(* IEC 61131-3 sources: ATCMcontrol_Engineering/src/Target/ATHW119/Libs/ATCM_System2, 31 files *)

(* ---- EVT_GetEvent.st ---- *)
(*
 * ATCMControl Embedded - System Library
 * ----------------------------------------------------------------------------
 *

 *)

(*[[
    UserURL= "ATCMfile:EVT_GetEvent.htm"
]]*)

(* EVT_GetEvent
 * ----------------------------------------------------------------------------
 * Gets the last event whiched caused the execution of the corresponding event
 * driven task.
 *
 * in   sTask       Task name.
 * out  uEvent      Last task execution event number.
 * ret              OK if successful else error number (see ErrNo.cst).
 *)
FUNCTION EVT_GetEvent : WORD

VAR_INPUT
    sTask  : STRING;
END_VAR

VAR_OUTPUT
    uEvent : INT;
END_VAR

inline{STDLIB(EVT_GetEvent)}

END_FUNCTION

(* ---- EVT_GetException.st ---- *)
(*
 * ATCMControl Embedded - System Library
 * ----------------------------------------------------------------------------
 *

 *)

(*[[
    UserURL= "ATCMfile:EVT_GetException.htm"
]]*)

(* EVT_GetException
 * ----------------------------------------------------------------------------
 * Gets the task number and exception number of the last raised task exception.
 * (To be used as an exception event handler.)
 *
 * out  uTask       Task index number of last exception.
 * out  ulException Exception number.
 * ret              OK if successful else error number (see ErrNo.cst).
 *)
FUNCTION EVT_GetException : WORD

VAR_OUTPUT
    uTask       : INT;
    ulException : DINT;
END_VAR

inline{STDLIB(EVT_GetException)}

END_FUNCTION

(* ---- EVT_Set.st ---- *)
(*
 * ATCMControl Embedded - System Library
 * ----------------------------------------------------------------------------
 *

 *)

(*[[
    UserURL= "ATCMfile:EVT_Set.htm"
]]*)

(* EVT_SET
 * ----------------------------------------------------------------------------
 * Sets a givent event.
 *
 * in   uEvent      Event to be set.
 * ret              OK if successful else error number (see ErrNo.cst).
 *)
FUNCTION EVT_Set : WORD

VAR_INPUT
    uEvent       : INT;
END_VAR

inline{STDLIB(EVT_Set)}

END_FUNCTION

(* ---- LD_Get.st ---- *)
(*
 * ATCMControl Embedded - System Library
 * ----------------------------------------------------------------------------
 *

 *)

FUNCTION LD_Get : WORD

(* Warning: This function is not thread safe. Calling this function from
 * different tasks for the same load type may cause unpredictable results!
 *)

VAR_INPUT
    LoadType    : WORD;         (* See SysLoad.cst for details.     *)
    TaskID      : UINT;         (* See SysLoad.cst for details.     *)
END_VAR

VAR_OUTPUT
    str         : STRING;
END_VAR

inline {STDLIB(LD_Get)}

END_FUNCTION

(* ---- MSG_SendToEng.st ---- *)
(*
 * ATCMControl Embedded - System Library
 * ----------------------------------------------------------------------------
 *

 *)

(*[[
    UserURL= "ATCMfile:MSG_SendToEng.htm"
]]*)

(* MSG_SendToEng
 * ----------------------------------------------------------------------------
 * Sends a message to the targets message view in the ATCMControl Engineering.
 *
 * in   sMsg        Message to send to the Engineering.
 *)
FUNCTION MSG_SendToEng

VAR_INPUT
    sMsg : STRING;
END_VAR

inline{STDLIB(MSG_SendToEng)}

END_FUNCTION

(* ---- MSG_Trace.st ---- *)
(*
 * ATCMControl Embedded - System Library
 * ----------------------------------------------------------------------------
 *

 *)

(*[[
    UserURL= "ATCMfile:MSG_Trace.htm"
]]*)

(* MSG_Trace
 * ----------------------------------------------------------------------------
 * Sends a message to the RTS trace device.
 *
 * in   sMsg        Message to trace.
 *)

FUNCTION MSG_Trace

VAR_INPUT
    sMsg : STRING;
END_VAR

inline{STDLIB(MSG_Trace)}

END_FUNCTION

(* ---- SFC_ResetToInitial.st ---- *)
(*
 * ATCMControl Embedded - System Library
 * ----------------------------------------------------------------------------
 *

 *)

(*[[
    UserURL= "ATCMfile:SFC_ResetToInitial.htm"
]]*)

(* SFC_ResetToInitial
 * ----------------------------------------------------------------------------
 * Resets the SFC logic.
 * in   bEnable         Reset only if TRUE.
 *)
FUNCTION SFC_ResetToInitial

VAR_INPUT
    bEnable : BOOL; (* reset only if bEnable = TRUE *)
END_VAR

inline
{
    push1        %1
    POPD_IN_1    __resetSFC
}

END_FUNCTION

(* ---- SYS_Coldstart.st ---- *)
(*
 * ATCMControl Embedded - System Library
 * ----------------------------------------------------------------------------
 *

 *)

(*[[
    UserURL= "ATCMfile:SYS_Coldstart.htm"
]]*)

(* SYS_Coldstart
 * ----------------------------------------------------------------------------
 * Executes a cold start of the ATCMControl Run Time System.
 *
 * ret              OK if successful else error number (see ErrNo.cst).
 *)
FUNCTION SYS_Coldstart : WORD

inline{STDLIB(SYS_Coldstart)}

END_FUNCTION

(* ---- SYS_Reboot.st ---- *)
(*
 * ATCMControl Embedded - System Library
 * ----------------------------------------------------------------------------
 *

 *)

(*[[
    UserURL= "ATCMfile:SYS_Reboot.htm"
]]*)

(* SYS_Reboot
 * ----------------------------------------------------------------------------
 * Reboots the controller hardware. (Only if supported on the corresponding
 * hardware environment!)
 *
 * ret              OK if successful else error number (see ErrNo.cst).
 *)
FUNCTION SYS_Reboot : WORD

inline{STDLIB(SYS_Reboot)}

END_FUNCTION

(* ---- SYS_RetainWrite.st ---- *)
(*
 * ATCMControl Embedded - System Library
 * ----------------------------------------------------------------------------
 *

 *)

(*[[
    UserURL= "ATCMfile:SYS_RetainWrite.htm"
]]*)

(* SYS_RetainWrite
 * ----------------------------------------------------------------------------
 * Writes the IEC retain segment to the file system. (Not supported on all
 * targets and only if no real physical retentive memory is available.)
 *
 * ret              OK if successful else error number (see ErrNo.cst).
 *)
FUNCTION SYS_RetainWrite : WORD

inline{STDLIB(SYS_RetainWrite)}

END_FUNCTION

(* ---- SYS_Warmstart.st ---- *)
(*
 * ATCMControl Embedded - System Library
 * ----------------------------------------------------------------------------
 *

 *)

(*[[
    UserURL= "ATCMfile:SYS_Warmstart.htm"
]]*)

(* SYS_Warmstart
 * ----------------------------------------------------------------------------
 * Executes a warm start of the ATCMControl Run Time System.
 *
 * ret              OK if successful else error number (see ErrNo.cst).
 *)
FUNCTION SYS_Warmstart : WORD

inline{STDLIB(SYS_Warmstart)}

END_FUNCTION

(* ---- TIM_Get.st ---- *)
(*
 * ATCMControl Embedded - System Library
 * ----------------------------------------------------------------------------
 *

 *)

(*[[
    UserURL= "ATCMfile:TIM_Get.htm"
]]*)

(* TSK_GetTime
 * ----------------------------------------------------------------------------
 * Gets the current system time.
 *
 * ret              Current system time.
 *)
FUNCTION TIM_Get : TIME

inline {STDLIB(TIM_Get)}

END_FUNCTION

(* ---- TSK_ClearError.st ---- *)
(*
 * ATCMControl Embedded - System Library
 * ----------------------------------------------------------------------------
 *

 *)

(*[[
    UserURL= "ATCMfile:TSK_ClearError.htm"
]]*)

(* TSK_ClearError
 * ----------------------------------------------------------------------------
 * Clears the task error number of the corresponding task.
 *
 * in   sTask       Task name.
 * ret              OK if successful else error number (see ErrNo.cst).
 *)
FUNCTION TSK_ClearError : WORD

VAR_INPUT
    sTask : STRING;
END_VAR

inline{STDLIB(TSK_ClearError)}

END_FUNCTION

(* ---- TSK_ClearStatistic.st ---- *)
(*
 * ATCMControl Embedded - System Library
 * ----------------------------------------------------------------------------
 *

 *)

(*[[
    UserURL= "ATCMfile:TSK_ClearStatistic.htm"
]]*)

(* TSK_ClearStatistic
 * ----------------------------------------------------------------------------
 * Clears the statistic information of the corresponding task.
 *
 * in   sTask       Task name.
 * ret              OK if successful else error number (see ErrNo.cst).
 *)
FUNCTION TSK_ClearStatistic : WORD

VAR_INPUT
    sTask    : STRING;
END_VAR

inline{STDLIB(TSK_ClearStatistic)}

END_FUNCTION

(* ---- TSK_Exception.st ---- *)
(*
 * ATCMControl Embedded - System Library
 * ----------------------------------------------------------------------------
 *

 *)

(*[[
    UserURL= "ATCMfile:TSK_Exception.htm"
]]*)

(* TSK_Exception
 * ----------------------------------------------------------------------------
 * Raises an exception in the current task.
 *
 * out  uExcepton   Exception index number.
 * ret              OK if successful else error number (see ErrNo.cst).
 *)
FUNCTION TSK_Exception : WORD

VAR_INPUT
    uException : INT;
END_VAR

inline{STDLIB(TSK_Exception)}

END_FUNCTION

(* ---- TSK_GetCount.st ---- *)
(*
 * ATCMControl Embedded - System Library
 * ----------------------------------------------------------------------------
 *

 *)

(*[[
    UserURL= "ATCMfile:TSK_GetCount.htm"
]]*)

(* TSK_GetCount
 * ----------------------------------------------------------------------------
 * Gets the number of tasks in the IEC project.
 *
 * ret              Number of tasks in project.
 *)
FUNCTION TSK_GetCount : INT

inline{STDLIB(TSK_GetCount)}

END_FUNCTION

(* ---- TSK_GetError.st ---- *)
(*
 * ATCMControl Embedded - System Library
 * ----------------------------------------------------------------------------
 *

 *)

(*[[
    UserURL= "ATCMfile:TSK_GetError.htm"
]]*)

(* TSK_GetError
 * ----------------------------------------------------------------------------
 * Gets the task error state of the corresponding task.
 *
 * in   sTask       Task name.
 * out  ulError     Task error state. (See ErrNo.cst for possible values.)
 * ret              OK if successful else error number (see ErrNo.cst).
 *)
FUNCTION TSK_GetError : WORD

VAR_INPUT
    sTask   : STRING;
END_VAR

VAR_OUTPUT
    ulError : DINT;
END_VAR

inline{STDLIB(TSK_GetError)}

END_FUNCTION

(* ---- TSK_GetInfo.st ---- *)
(*
 * ATCMControl Embedded - System Library
 * ----------------------------------------------------------------------------
 *

 *)

(*[[
    UserURL= "ATCMfile:TSK_GetInfo.htm"
]]*)

(* TSK_GetInfo
 * ----------------------------------------------------------------------------
 * Gets the task information structure of the corresponding task.
 *
 * in   sTask       Task name.
 * out  TaskInfo    Task information structure of task.
 * ret              OK if successful else error number (see ErrNo.cst).
 *)
FUNCTION TSK_GetInfo : WORD

VAR_INPUT
    sTask    : STRING;
END_VAR

VAR_OUTPUT
    TaskInfo : TSK_INFO;
END_VAR

inline{STDLIB(TSK_GetInfo)}

END_FUNCTION

(* ---- TSK_GetMyName.st ---- *)
(*
 * ATCMControl Embedded - System Library
 * ----------------------------------------------------------------------------
 *

 *)

(*[[
    UserURL= "ATCMfile:TSK_GetMyName.htm"
]]*)

(* TSK_GetMyName
 * ----------------------------------------------------------------------------
 * Gets the name of the calling task.
 *
 * ret              Name of the calling task.
 *)
FUNCTION TSK_GetMyName : STRING

inline{STDLIB(TSK_GetMyName)}

END_FUNCTION

(* ---- TSK_GetMyNumber.st ---- *)
(*
 * ATCMControl Embedded - System Library
 * ----------------------------------------------------------------------------
 *

 *)

(*[[
    UserURL= "ATCMfile:TSK_GetMyNumber.htm"
]]*)

(* TSK_GetMyNumber
 * ----------------------------------------------------------------------------
 * Gets the index number of the calling task.
 *
 * ret              Task index number of calling task.
 *)
FUNCTION TSK_GetMyNumber : INT

inline{STDLIB(TSK_GetMyNumber)}

END_FUNCTION

(* ---- TSK_GetName.st ---- *)
(*
 * ATCMControl Embedded - System Library
 * ----------------------------------------------------------------------------
 *

 *)

(*[[
    UserURL= "ATCMfile:TSK_GetName.htm"
]]*)

(* TSK_GetName
 * ----------------------------------------------------------------------------
 * Gets the task name of a task identified by its task index number.
 *
 * in   uTask       Task index number.
 * out  sTask       Task name.
 * ret              OK if successful else error number (see ErrNo.cst).
 *)
FUNCTION TSK_GetName : WORD

VAR_INPUT
    uTask   : INT;
END_VAR

VAR_OUTPUT
    sTask   : STRING;
END_VAR

inline{STDLIB(TSK_GetName)}

END_FUNCTION

(* ---- TSK_GetState.st ---- *)
(*
 * ATCMControl Embedded - System Library
 * ----------------------------------------------------------------------------
 *

 *)

(*[[
    UserURL= "ATCMfile:TSK_GetState.htm"
]]*)

(* TSK_GetState
 * ----------------------------------------------------------------------------
 * Gets the task state of the corresponding task.
 *
 * in   sTask       Task name.
 * out  ulState     Task state. (See System2.cst for possible values.)
 * ret              OK if successful else error number (see ErrNo.cst).
 *)
FUNCTION TSK_GetState : WORD

VAR_INPUT
    sTask   : STRING;
END_VAR

VAR_OUTPUT
    ulState : DINT;
END_VAR

inline{STDLIB(TSK_GetState)}

END_FUNCTION

(* ---- TSK_GetStatistic.st ---- *)
(*
 * ATCMControl Embedded - System Library
 * ----------------------------------------------------------------------------
 *

 *)

(*[[
    UserURL= "ATCMfile:TSK_GetStatistic.htm"
]]*)

(* TSK_GetStatistic
 * ----------------------------------------------------------------------------
 * Gets statistic information of the corresponding task.
 *
 * in   sTask       Task name.
 * out  TaskStat    Task statistics of corresponding task.
 * ret              OK if successful else error number (see ErrNo.cst).
 *)
FUNCTION TSK_GetStatistic : WORD

VAR_INPUT
    sTask    : STRING;
END_VAR

VAR_OUTPUT
    TaskStat : TSK_Stat;
END_VAR

inline{STDLIB(TSK_GetStatistic)}

END_FUNCTION

(* ---- TSK_Start.st ---- *)
(*
 * ATCMControl Embedded - System Library
 * ----------------------------------------------------------------------------
 *

 *)

(*[[
    UserURL= "ATCMfile:TSK_Start.htm"
]]*)

(* TSK_Start
 * ----------------------------------------------------------------------------
 * Starts the corresponding task.
 *
 * in   sTask       Task name.
 * ret              OK if successful else error number (see ErrNo.cst).
 *)
FUNCTION TSK_Start : WORD

VAR_INPUT
    sTask : STRING;
END_VAR

inline{STDLIB(TSK_Start)}

END_FUNCTION

(* ---- TSK_Stop.st ---- *)
(*
 * ATCMControl Embedded - System Library
 * ----------------------------------------------------------------------------
 *

 *)

(*[[
    UserURL= "ATCMfile:TSK_Stop.htm"
]]*)

(* TSK_Stop
 * ----------------------------------------------------------------------------
 * Stops the corresponding task.
 *
 * in   sTask       Task name.
 * ret              OK if successful else error number (see ErrNo.cst).
 *)
FUNCTION TSK_Stop : WORD

VAR_INPUT
    sTask : STRING;
END_VAR

inline{STDLIB(TSK_Stop)}

END_FUNCTION

(* ---- WD_Disable.st ---- *)
(*
 * ATCMControl Embedded - System Library
 * ----------------------------------------------------------------------------
 *

 *)

(*[[
    UserURL= "ATCMfile:WD_Disable.htm"
]]*)

(* WD_Disable
 * ----------------------------------------------------------------------------
 * Disables (cancels) a watchdog for the corresponding task.
 *
 * in   sTask       Task name.
 * ret              OK if successful else error number (see ErrNo.cst).
 *)
FUNCTION WD_Disable : WORD

VAR_INPUT
    sTask : STRING;
END_VAR

inline{STDLIB(WD_Disable)}

END_FUNCTION

(* ---- WD_Enable.st ---- *)
(*
 * ATCMControl Embedded - System Library
 * ----------------------------------------------------------------------------
 *

 *)

(*[[
    UserURL= "ATCMfile:WD_Enable.htm"
]]*)

(* WD_Enable
 * ----------------------------------------------------------------------------
 * Enables (start) the watchdog for the corresponding task. If the watchdog
 * doesn't already exist, a new watchdog is created.
 *
 * in   sTask       Task name.
 * ret              OK if successful else error number (see ErrNo.cst).
 *)
FUNCTION WD_Enable : WORD

VAR_INPUT
    sTask    : STRING;
END_VAR

inline{STDLIB(WD_Enable)}

END_FUNCTION

(* ---- WD_GetTrigger.st ---- *)
(*
 * ATCMControl Embedded - System Library
 * ----------------------------------------------------------------------------
 *

 *)

(*[[
    UserURL= "ATCMfile:WD_GetTrigger.htm"
]]*)

(* WD_GetTrigger
 * ----------------------------------------------------------------------------
 * Gets the watchdog trigger level and the actual watchdog trigger count of
 * the corresponding task.
 *
 * in   sTask       Task name.
 * out  WDTrigger   Watchdog trigger level.
 * out  WDCount     Actual watchdog trigger count.
 * ret              OK if successful else error number (see ErrNo.cst).
 *)
FUNCTION WD_GetTrigger : WORD

VAR_INPUT
    sTask     : STRING;
END_VAR

VAR_OUTPUT
    WDTrigger   : UDINT;
    WDCount     : UDINT;
END_VAR

inline{STDLIB(WD_GetTrigger)}

END_FUNCTION

(* ---- WD_IsEnabled.st ---- *)
(*
 * ATCMControl Embedded - System Library
 * ----------------------------------------------------------------------------
 *

 *)

(*[[
    UserURL= "ATCMfile:WD_IsEnabled.htm"
]]*)

(* WD_IsEnabled
 * ----------------------------------------------------------------------------
 * Gets the watchdog state (enabled / disabled) for the given task.
 *
 * in   sTask       Task name.
 * ou   bEnabled    Watchdog state (enabled / disabled).
 * ret              OK if successful else error number (see ErrNo.cst).
 *)
FUNCTION WD_IsEnabled : WORD

VAR_INPUT
    sTask    : STRING;
END_VAR

VAR_OUTPUT
    bEnabled : BOOL;
END_VAR

inline{STDLIB(WD_IsEnabled)}

END_FUNCTION

(* ---- WD_SetTrigger.st ---- *)
(*
 * ATCMControl Embedded - System Library
 * ----------------------------------------------------------------------------
 *

 *)

(*[[
    UserURL= "ATCMfile:WD_SetTrigger.htm"
]]*)

(* WD_SetTrigger
 * ----------------------------------------------------------------------------
 * Sets the watchdog trigger level of the corresponding task.
 *
 * in   sTask       Task name.
 * in   WDTrigger   Watchdog trigger level.
 * ret              OK if successful else error number (see ErrNo.cst).
 *)
FUNCTION WD_SetTrigger : WORD

VAR_INPUT
    sTask       : STRING;
END_VAR

VAR_INPUT
    WDTrigger   : UDINT;
END_VAR

inline{STDLIB(WD_SetTrigger)}

END_FUNCTION

(* ---- SYS_TraceStat.st ---- *)
(*
 * ATCMControl Embedded - System Library
 * ----------------------------------------------------------------------------
 *

 *)

(*[[
]]*)

(* SYS_TraceStat
 * ----------------------------------------------------------------------------
 * Traces the actual load statistics to the Engineering.
 * Warning: This function block is not thread safe and creates a significant
 * amount of processor load itself.
 *
 * in  tCycle       Cycle time.
 *)
FUNCTION_BLOCK SYS_TraceStat

VAR_INPUT
    tCycle  : TIME := t#5s;
END_VAR
VAR
    tLast   : TIME;
    tNow    : TIME;

    wRes    : WORD;
    str     : STRING;
END_VAR

    tNow := Tim_Get();

    if tNow < tLast + tCycle then
        return;
    end_if;

    tLast := tNow;

    wRes := LD_Get(LOAD_LOAD_AVERAGE, 0, str);
    if wRes = OK then MSG_SendToEng(str); end_if;

    wRes := LD_Get(LOAD_CPU_SYSTEM, 0, str);
    if wRes = OK then MSG_SendToEng(str); end_if;

    wRes := LD_Get(LOAD_CPU_IEC, 0, str);
    if wRes = OK then MSG_SendToEng(str); end_if;

    wRes := LD_Get(LOAD_CPU_RTS, 0, str);
    if wRes = OK then MSG_SendToEng(str); end_if;

    MSG_SendToEng('--------------------------------------------------------------');

END_FUNCTION_BLOCK
